FUNCTION_BLOCK E_CALIBRATE_3P (* Event-driven 3-point calibration for joysticks (Min, Mid, Max) *)
  (* Standard: 61499-1 *)
  (* Version 1.0, 2026-06-01, Meisterschulen am Ostbahnhof *)
  PACKAGE OSCAT::Basic::POUs::Engineering::measurements;
  (* Documentation:
  Formula
    Y = piecewise linear interpolation between stored calibration points Calibration (3-Point)
    - Min (EI_MIN): Move joystick to minimum position, fire EI_MIN
   X_MIN := X → stores current raw value as Min point
   - Mid (EI_MID): Move joystick to center, fire EI_MID
   X_MID := X → stores current raw value as Mid point (center)
   - Max (EI_MAX): Move joystick to maximum position, fire EI_MAX
   X_MAX := X → stores current raw value as Max point
    Note: The calibration points can be calibrated in any order and can be repeated individually.
   Output Calculation
    - If X < X_MID: linear interpolation between (X_MIN, MIN_REF) and (X_MID, MID_REF)
   - If X >= X_MID: linear interpolation between (X_MID, MID_REF) and (X_MAX, MAX_REF)
   - Output is clipped to MIN_REF..MAX_REF
    ECC State Machine
    START --REQ--> REQ --1--> START       (normal operation) START -EI_MIN-> C_MIN --1--> START    (calibrate minimum) START -EI_MID-> C_MID --1--> START    (calibrate center) START -EI_MAX-> C_MAX --1--> START    (calibrate maximum) All calibration events are independently accessible from the START state – no enforced order.
   Example
   Scenario: Joystick with center drift. Raw range 0..1000, desired output -100..0..100.
      Step |  Action |  Result |  
    1 |  Move joystick to min, fire EI_MIN |  X_MIN = 50 (drifted from ideal 0) |  
    2 |  Move joystick to center, fire EI_MID |  X_MID = 520 (drifted from ideal 500) |  
    3 |  Move joystick to max, fire EI_MAX |  X_MAX = 980 (drifted from ideal 1000) |  
     Output: Interpolated between MIN_REF=-100, MID_REF=0, MAX_REF=100 with clipping.
  *)
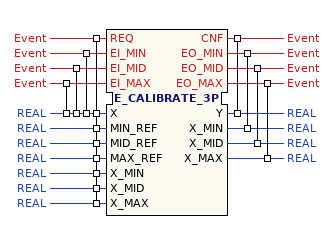
  EVENT_INPUT
    REQ WITH X, MIN_REF, MID_REF, MAX_REF, X_MIN, X_MID, X_MAX; (* Normal Execution Request *)
    EI_MIN WITH X; (* Calibrate Min Point *)
    EI_MID WITH X; (* Calibrate Mid Point (Center) *)
    EI_MAX WITH X; (* Calibrate Max Point *)
  END_EVENT
  EVENT_OUTPUT
    CNF WITH Y; (* Execution Confirmation *)
    EO_MIN WITH X_MIN; (* Min Calibration Confirmed *)
    EO_MID WITH X_MID; (* Mid Calibration Confirmed *)
    EO_MAX WITH X_MAX; (* Max Calibration Confirmed *)
  END_EVENT
  VAR_INPUT
    X : REAL; (* Raw Input *)
    MIN_REF : REAL := 0.0; (* Target value for Min *)
    MID_REF : REAL := 50.0; (* Target value for Mid *)
    MAX_REF : REAL := 100.0; (* Target value for Max *)
  END_VAR
  VAR_OUTPUT
    Y : REAL; (* Calibrated Output *)
  END_VAR
  VAR_IN_OUT
    X_MIN : REAL := 0.0; (* Stored Min Value *)
    X_MID : REAL := 50.0; (* Stored Mid Value *)
    X_MAX : REAL := 100.0; (* Stored Max Value *)
  END_VAR
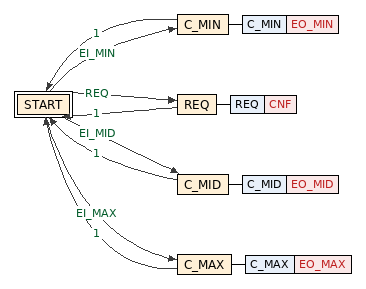
  EC_STATES
    START;
    REQ : REQ -> CNF;
    C_MIN : C_MIN -> EO_MIN;
    C_MID : C_MID -> EO_MID;
    C_MAX : C_MAX -> EO_MAX;
  END_STATES
  EC_TRANSITIONS
    START TO REQ := REQ;
    REQ TO START := 1;
    START TO C_MIN := EI_MIN;
    C_MIN TO START := 1;
    START TO C_MID := EI_MID;
    C_MID TO START := 1;
    START TO C_MAX := EI_MAX;
    C_MAX TO START := 1;
  END_TRANSITIONS
  ALGORITHM REQ IN ST:
(* calculate output *)
IF X < X_MID THEN
	IF X_MID > X_MIN THEN
		Y := MIN_REF + (X - X_MIN) * (MID_REF - MIN_REF) / (X_MID - X_MIN);
	ELSE
		Y := MIN_REF;
	END_IF;
ELSE
	IF X_MAX > X_MID THEN
		Y := MID_REF + (X - X_MID) * (MAX_REF - MID_REF) / (X_MAX - X_MID);
	ELSE
		Y := MID_REF;
	END_IF;
END_IF;

(* clipping *)
IF Y < MIN_REF THEN
	Y := MIN_REF;
ELSIF Y > MAX_REF THEN
	Y := MAX_REF;
END_IF;
  END_ALGORITHM
  ALGORITHM C_MIN IN ST:
(* store current raw input as Min calibration point *)
X_MIN := X;
  END_ALGORITHM
  ALGORITHM C_MID IN ST:
(* store current raw input as Mid calibration point (center) *)
X_MID := X;
  END_ALGORITHM
  ALGORITHM C_MAX IN ST:
(* store current raw input as Max calibration point *)
X_MAX := X;
  END_ALGORITHM
END_FUNCTION_BLOCK
